// LS Electric XG5000 project: asdfgh
// PLC LSPLC

PROGRAM NewProgram (task: 스캔 프로그램)

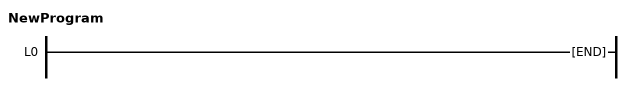
; L0
END